KUKA KRL data list: A43_global.dat

&ACCESS RV
&COMMENT V_1_4_0
&PARAM DISKPATH = KRC:\R1\BMW_App
&REL 4
DEFDAT A43_global PUBLIC
;********************************
;Date: 17.09.2021
;Programmer: AIUT
;Description: Global positions
;********************************


ENDDAT
